(* Logix 5000 project; controller Tekno_ASRS vendor 1 type 14 code 147 rev 20.11; software revision 20.01; part 3 of 4 *)
(* tags used below, declared in another part *)
   AutoMode : BOOL;
   AAxis : AXIS_CIP_DRIVE;
   AAxisJog : MOTION_INSTRUCTION;
   AAxisMAM : MOTION_INSTRUCTION;
   AAxisMove : BOOL;
   AAxisOn : MOTION_INSTRUCTION;
   AAxisSODelay : TIMER;
   AAxisStop : MOTION_INSTRUCTION;
   ABayPos : DINT;
   ABGrid : Position[100,20];
   AgridLoc : DINT;
   AGVatDP : ALIAS FOR StationaryIO:1:I.3;
   AGVatPU : ALIAS FOR StationaryIO:1:I.2;
   AGVDP : BOOL;
   AGVok2LvDP : ALIAS FOR StationaryIO:8:O.0;
   AGVok2LvPU : ALIAS FOR StationaryIO:8:O.1;
   AGVPU : BOOL;
   AGVPUHoldTmr : TIMER;
   AInc : DINT;
   AllowSynchAB : BOOL;
   APitch : REAL;
   APos : REAL;
   ARange : REAL;
   AReq : DINT;
   AReqPos : REAL;
   ASRSMCR : BOOL;
   AStart : REAL;
   BAxis : AXIS_CIP_DRIVE;
   BAxisJog : MOTION_INSTRUCTION;
   BAxisMAM : MOTION_INSTRUCTION;
   BAxisMove : BOOL;
   BAxisOn : MOTION_INSTRUCTION;
   BAxisSODelay : TIMER;
   BAxisStop : MOTION_INSTRUCTION;
   BBayPos : DINT;
   BgridLoc : DINT;
   BInc : DINT;
   BPitch : REAL;
   BPos : REAL;
   BRange : DINT;
   BReq : DINT;
   BReqPos : REAL;
   BStart : REAL;
   CCoordSetup : BOOL;
   CfgEnd : BayPos;
   CfgStrt : BayPos;
   CfgTtlAAxis : DINT;
   CfgTtlBAxis : DINT;
   CFinalPos : DINT;
   CGridLoc : DINT;
   CHomePos : DINT;
   Configuration : Configuration;
   CPosHighLim : DINT;
   CPosLowLim : DINT;
   CPosSpeed2Tol : DINT;
   CPosTolerance : DINT;
   CReq : DINT;
   CReqPos : DINT;
   CurrentAPos : DINT;
   CurrentBPos : DINT;
   CurrentCPos : DINT;
   CurrentTask : Task;
   DepositReq : BOOL;
   FootSwitch : ALIAS FOR ShuttleIO:9:I.Pt04Data;
   HMI_Commands : HMI_Commands;
   HomeSpatula : BOOL;
   JogAAxisEn : BOOL;
   JogActive : BOOL;
   JogARev : BOOL;
   JogBAxisEn : BOOL;
   JogBFwd : BOOL;
   JogBRev : BOOL;
   JogConfiguration : Configuration;
   JogEnabled : BOOL;
   JogReleaseSBrk : BOOL;
   Last : DINT;
   LastAAxErr : DINT;
   LastAAxExErr : DINT;
   LastMessageReceiveSequence : DINT;
   LoadTask : Task;
   LockRelease : ALIAS FOR StationaryIO:7:I.Pt04Data;
   ManOnBoard : ALIAS FOR ShuttleIO:5:O.5;
   MatrixSetup : BOOL;
   MaxA : DINT;
   MaxB : DINT;
   MoveComplete : BOOL;
   MoveInProcess : BOOL;
   MoveReady : BOOL;
   MoveRequested : BOOL;
   MoveSafetyEnable : BOOL;
   MsgTimer : TIMER;
   MtrEndDsbleZn : REAL;
   OperatorDN : BOOL;
   PnlEndDsbleZn : REAL;
   PorDInProc : BOOL;
   PorDStepTemp : BOOL;
   PorDStop : BOOL;
   PositionFlt : BOOL;
   ReceiveMessage : Messaging;
   ReleaseSpatBrk : BOOL;
   SendMessage : Messaging;
   SendMessageCommand : MESSAGE;
   SpatSimHome : BOOL;
   SpatulaBrake : ALIAS FOR ShuttleIO:5:O.6;
   SpatulaExtendComp : BOOL;
   SpatulaExtended : BOOL;
   SpatulaHome : ALIAS FOR ShuttleIO:2:I.4;
   SpatulaStopped : BOOL;
   SUIndPos : BOOL;
   TaskFIFO : CONTROL;
   TaskFile : Task[100];
   TaskInProcess : BOOL;
   TestStop : BOOL;
   XAccuracy : REAL;
   XAxisMtrSideEOT : ALIAS FOR ShuttleIO:2:I.6;
   XAxisPnlSideEOT : ALIAS FOR ShuttleIO:2:I.7;
   XHighLimit : REAL;
   XLftTempDint1 : DINT;
   XLftTempDint2 : DINT;
   XLftTempFloat1 : REAL;
   XLftTempFloat2 : REAL;
   XLftTempFloat3 : REAL;
   XLowLimit : REAL;
   XRgtTempDint1 : DINT;
   XRgtTempDint2 : REAL;
   XRgtTempFloat1 : REAL;
   XRgtTempFloat2 : REAL;
   XRgtTempFloat3 : REAL;
   XStCalMode : ALIAS FOR StationaryIO:5:O.Data[0].0;
   XStLftSignRun : ALIAS FOR StationaryIO:5:I.Data[7].7;
   XStrain : Strain;
   XStrainHigh : DINT;
   XStrainLow : DINT;
   XStRtSignRun : ALIAS FOR StationaryIO:5:I.Data[11].7;
   XStRunMode : ALIAS FOR StationaryIO:5:O.Data[0].1;
   XTensionOK : BOOL;
   ZAccuracy : REAL;
   ZAxisDnEOT : ALIAS FOR ShuttleIO:1:I.1;
   ZAxisUpEOT : ALIAS FOR ShuttleIO:1:I.0;
   ZForeStCalMode : ALIAS FOR ShuttleIO:3:O.Data[0].0;
   ZForeStrain : Strain;
   ZForeStRunMode : ALIAS FOR ShuttleIO:3:O.Data[0].1;
   ZHighLimit : REAL;
   ZLBindTmr : TIMER;
   ZLFault : BOOL;
   ZLowLimit : REAL;
   ZLsDisengaged : BOOL;
(* MainProgram, continued *)

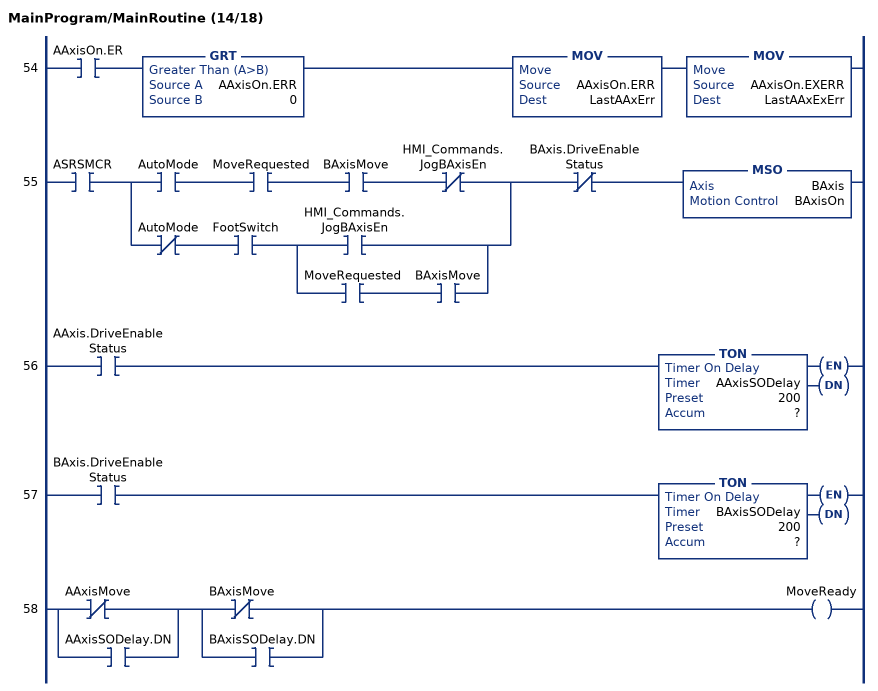
   [picture p24: MainProgram/MainRoutine rungs 54-58]
   54: XIC(AAxisOn.ER)GRT(AAxisOn.ERR,0)MOV(AAxisOn.ERR,LastAAxErr)MOV(AAxisOn.EXERR,LastAAxExErr);
   55: XIC(ASRSMCR)[XIC(AutoMode) XIC(MoveRequested) XIC(BAxisMove) XIO(HMI_Commands.JogBAxisEn) ,XIO(AutoMode) XIC(FootSwitch) [XIC(HMI_Commands.JogBAxisEn) ,XIC(MoveRequested) XIC(BAxisMove) ] ]XIO(BAxis.DriveEnableStatus)MSO(BAxis,BAxisOn);
   56: XIC(AAxis.DriveEnableStatus)TON(AAxisSODelay,?,?);
   57: XIC(BAxis.DriveEnableStatus)TON(BAxisSODelay,?,?);
   58: [XIO(AAxisMove) ,XIC(AAxisSODelay.DN) ][XIO(BAxisMove) ,XIC(BAxisSODelay.DN) ]OTE(MoveReady);
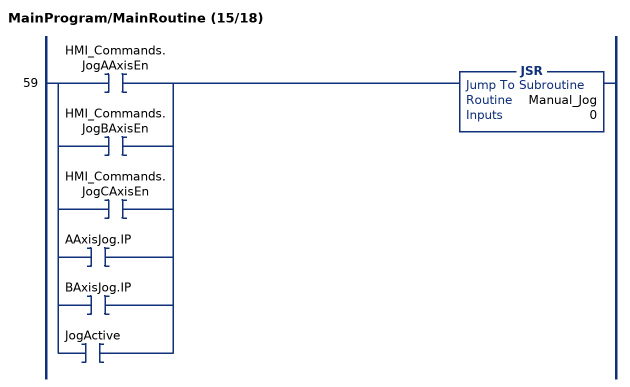
   59: [XIC(HMI_Commands.JogAAxisEn) ,XIC(HMI_Commands.JogBAxisEn) ,XIC(HMI_Commands.JogCAxisEn) ,XIC(AAxisJog.IP) ,XIC(BAxisJog.IP) ,XIC(JogActive) ]JSR(Manual_Jog,0);
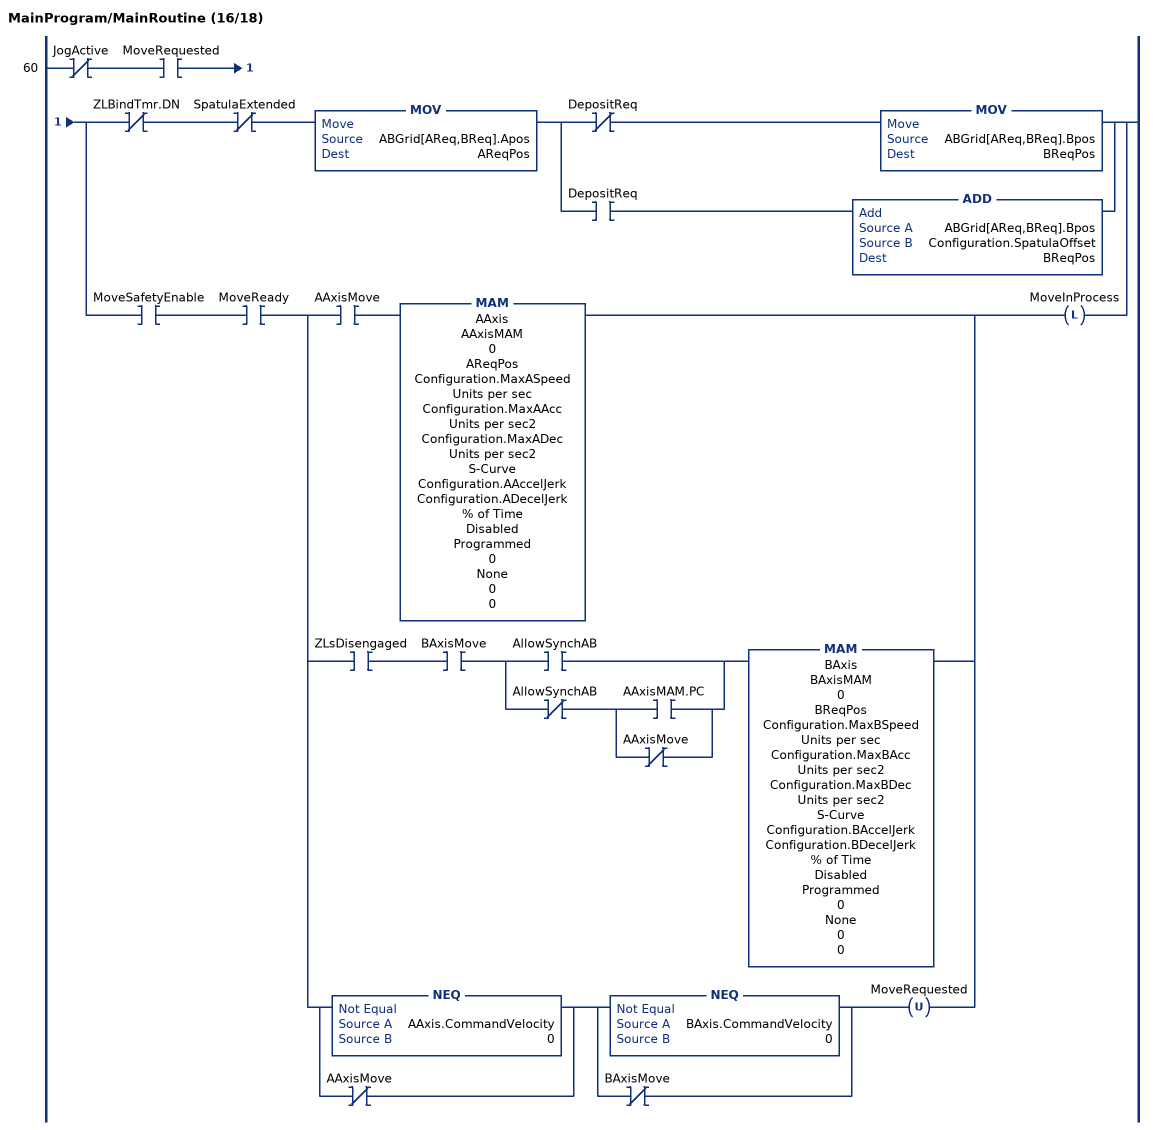
   60: XIO(JogActive)XIC(MoveRequested)[XIO(ZLBindTmr.DN) XIO(SpatulaExtended) MOV(ABGrid[AReq,BReq].Apos,AReqPos) [XIO(DepositReq) MOV(ABGrid[AReq,BReq].Bpos,BReqPos) ,XIC(DepositReq) ADD(ABGrid[AReq,BReq].Bpos,Configuration.SpatulaOffset,BReqPos) ] ,XIC(MoveSafetyEnable) XIC(MoveReady) [XIC(AAxisMove) MAM(AAxis,AAxisMAM,0,AReqPos,Configuration.MaxASpeed,Units per sec,Configuration.MaxAAcc,Units per sec2,Configuration.MaxADec,Units per sec2,S-Curve,Configuration.AAccelJerk,Configuration.ADecelJerk,% of Time,Disabled,Programmed,0,None,0,0) ,XIC(ZLsDisengaged) XIC(BAxisMove) [XIC(AllowSynchAB) ,XIO(AllowSynchAB) [XIC(AAxisMAM.PC) ,XIO(AAxisMove) ] ] MAM(BAxis,BAxisMAM,0,BReqPos,Configuration.MaxBSpeed,Units per sec,Configuration.MaxBAcc,Units per sec2,Configuration.MaxBDec,Units per sec2,S-Curve,Configuration.BAccelJerk,Configuration.BDecelJerk,% of Time,Disabled,Programmed,0,None,0,0) ,[NEQ(AAxis.CommandVelocity,0) ,XIO(AAxisMove) ] [NEQ(BAxis.CommandVelocity,0) ,XIO(BAxisMove) ] OTU(MoveRequested) ] OTL(MoveInProcess) ];
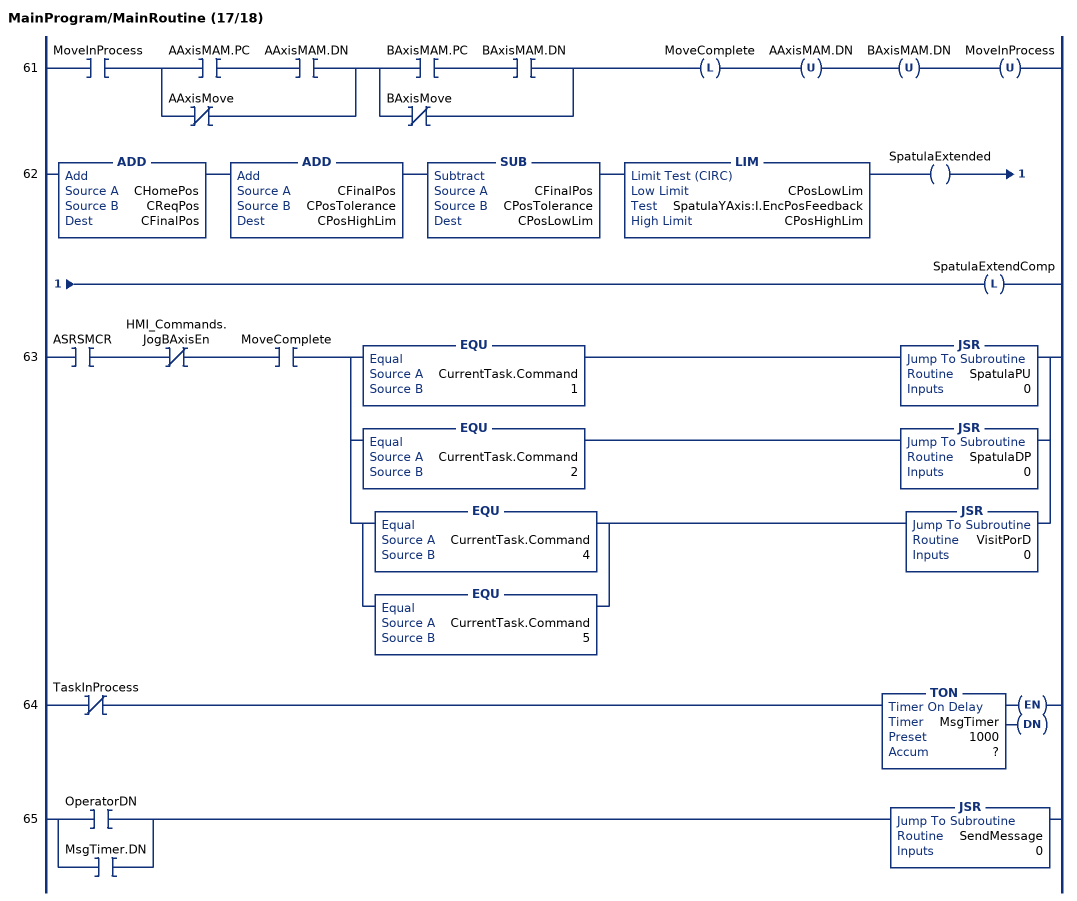
   61: XIC(MoveInProcess)[XIC(AAxisMAM.PC) XIC(AAxisMAM.DN) ,XIO(AAxisMove) ][XIC(BAxisMAM.PC) XIC(BAxisMAM.DN) ,XIO(BAxisMove) ]OTL(MoveComplete)OTU(AAxisMAM.DN)OTU(BAxisMAM.DN)OTU(MoveInProcess);
   62: ADD(CHomePos,CReqPos,CFinalPos)ADD(CFinalPos,CPosTolerance,CPosHighLim)SUB(CFinalPos,CPosTolerance,CPosLowLim)LIM(CPosLowLim,SpatulaYAxis:I.EncPosFeedback,CPosHighLim)OTE(SpatulaExtended)OTL(SpatulaExtendComp);
   63: XIC(ASRSMCR)XIO(HMI_Commands.JogBAxisEn)XIC(MoveComplete)[EQU(CurrentTask.Command,1) JSR(SpatulaPU,0) ,EQU(CurrentTask.Command,2) JSR(SpatulaDP,0) ,[EQU(CurrentTask.Command,4) ,EQU(CurrentTask.Command,5) ] JSR(VisitPorD,0) ];
   64: XIO(TaskInProcess)TON(MsgTimer,?,?);
   65: [XIC(OperatorDN) ,XIC(MsgTimer.DN) ]JSR(SendMessage,0);
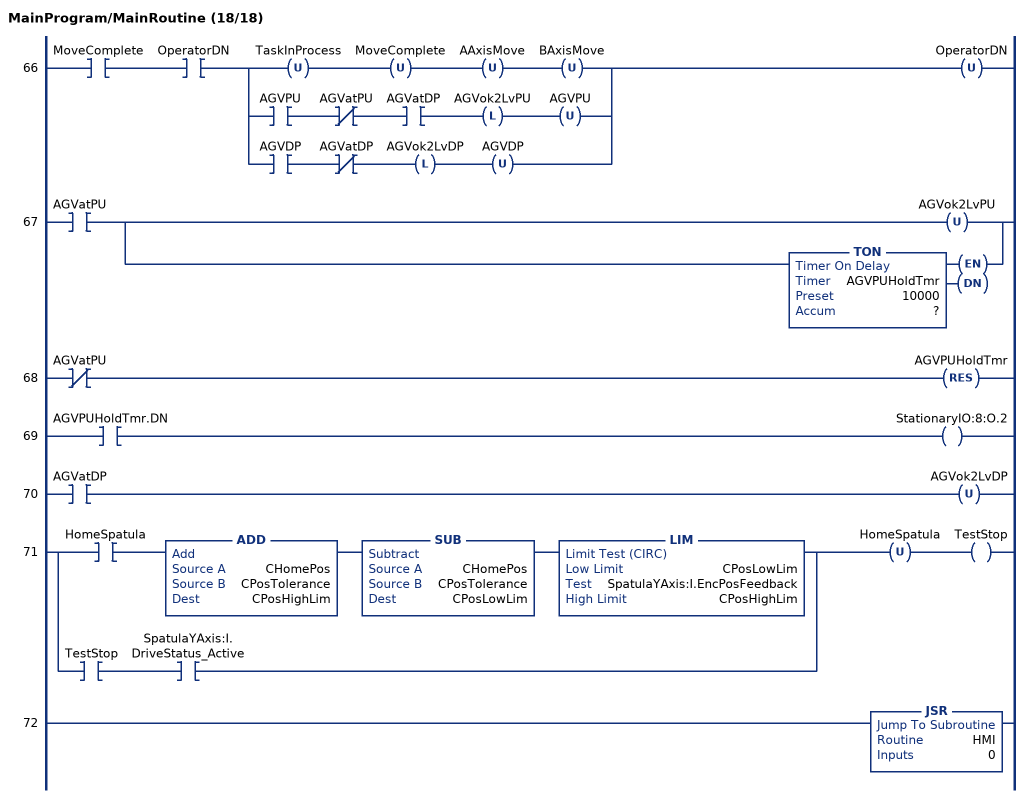
   66: XIC(MoveComplete)XIC(OperatorDN)[OTU(TaskInProcess) OTU(MoveComplete) OTU(AAxisMove) OTU(BAxisMove) ,XIC(AGVPU) XIO(AGVatPU) XIC(AGVatDP) OTL(AGVok2LvPU) OTU(AGVPU) ,XIC(AGVDP) XIO(AGVatDP) OTL(AGVok2LvDP) OTU(AGVDP) ]OTU(OperatorDN);
   67: XIC(AGVatPU)[OTU(AGVok2LvPU) ,TON(AGVPUHoldTmr,?,?) ];
   68: XIO(AGVatPU)RES(AGVPUHoldTmr);
   69: XIC(AGVPUHoldTmr.DN)OTE(StationaryIO:8:O.2);
   70: XIC(AGVatDP)OTU(AGVok2LvDP);
   71: [XIC(HomeSpatula) ADD(CHomePos,CPosTolerance,CPosHighLim) SUB(CHomePos,CPosTolerance,CPosLowLim) LIM(CPosLowLim,SpatulaYAxis:I.EncPosFeedback,CPosHighLim) ,XIC(TestStop) XIC(SpatulaYAxis:I.DriveStatus_Active) ]OTU(HomeSpatula)OTE(TestStop);
   72: JSR(HMI,0);
END_ROUTINE

ROUTINE Manual_Jog   (* ladder *)
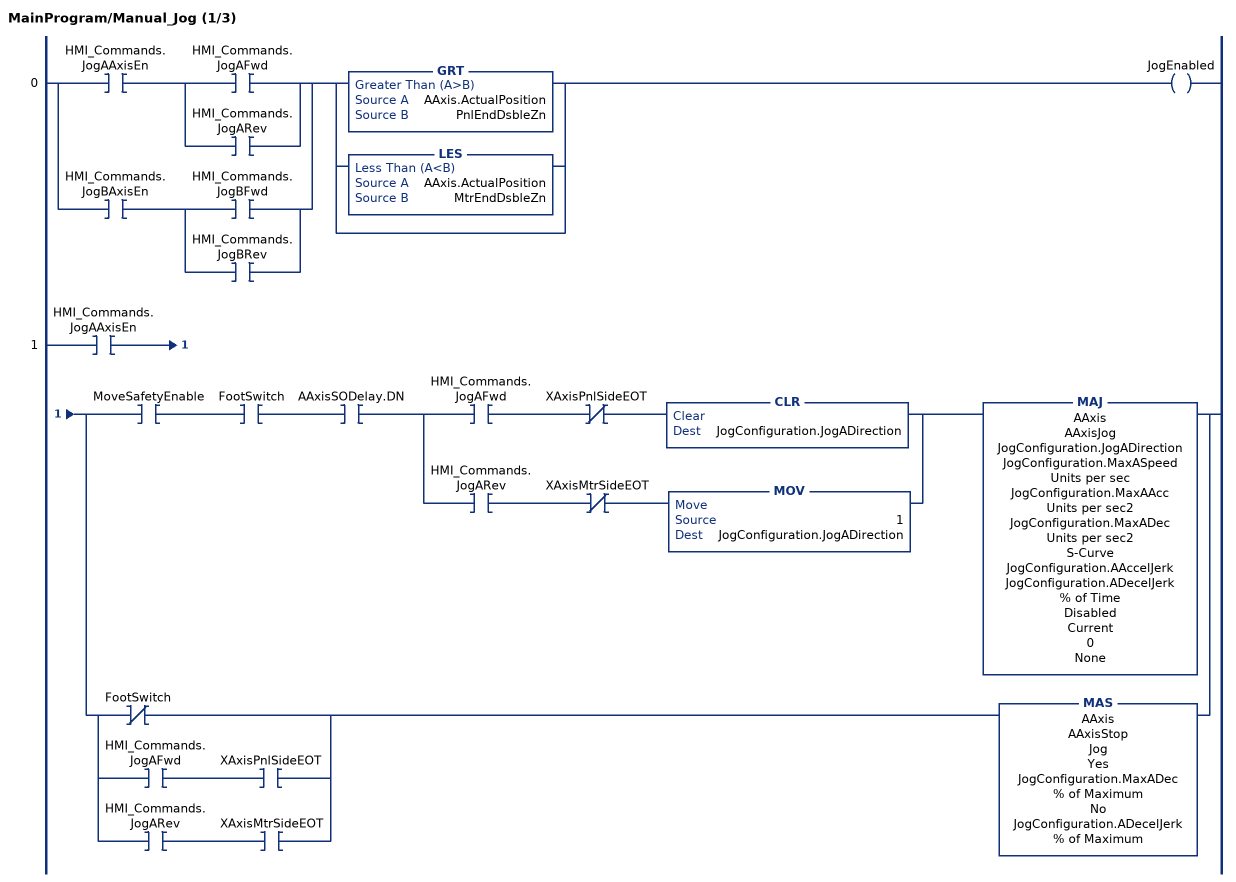
   0: [XIC(HMI_Commands.JogAAxisEn) [XIC(HMI_Commands.JogAFwd) ,XIC(HMI_Commands.JogARev) ] ,XIC(HMI_Commands.JogBAxisEn) [XIC(HMI_Commands.JogBFwd) ,XIC(HMI_Commands.JogBRev) ] ][GRT(AAxis.ActualPosition,PnlEndDsbleZn) ,LES(AAxis.ActualPosition,MtrEndDsbleZn) ,]OTE(JogEnabled);
   1: XIC(HMI_Commands.JogAAxisEn)[XIC(MoveSafetyEnable) XIC(FootSwitch) XIC(AAxisSODelay.DN) [XIC(HMI_Commands.JogAFwd) XIO(XAxisPnlSideEOT) CLR(JogConfiguration.JogADirection) ,XIC(HMI_Commands.JogARev) XIO(XAxisMtrSideEOT) MOV(1,JogConfiguration.JogADirection) ] MAJ(AAxis,AAxisJog,JogConfiguration.JogADirection,JogConfiguration.MaxASpeed,Units per sec,JogConfiguration.MaxAAcc,Units per sec2,JogConfiguration.MaxADec,Units per sec2,S-Curve,JogConfiguration.AAccelJerk,JogConfiguration.ADecelJerk,% of Time,Disabled,Current,0,None) ,[XIO(FootSwitch) ,XIC(HMI_Commands.JogAFwd) XIC(XAxisPnlSideEOT) ,XIC(HMI_Commands.JogARev) XIC(XAxisMtrSideEOT) ] MAS(AAxis,AAxisStop,Jog,Yes,JogConfiguration.MaxADec,% of Maximum,No,JogConfiguration.ADecelJerk,% of Maximum) ];
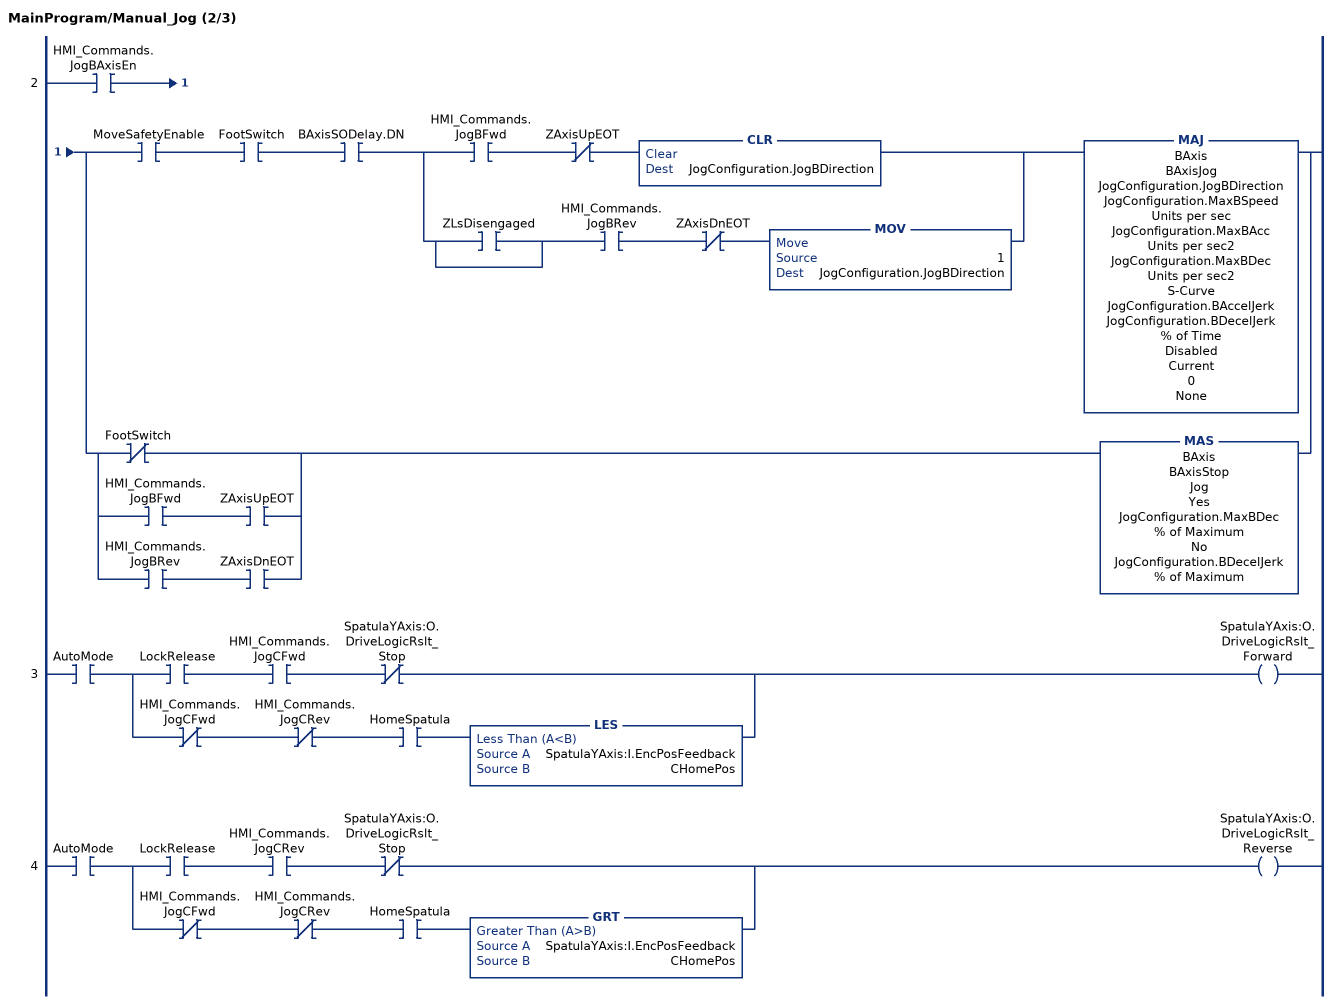
   2: XIC(HMI_Commands.JogBAxisEn)[XIC(MoveSafetyEnable) XIC(FootSwitch) XIC(BAxisSODelay.DN) [XIC(HMI_Commands.JogBFwd) XIO(ZAxisUpEOT) CLR(JogConfiguration.JogBDirection) ,[XIC(ZLsDisengaged) ,] XIC(HMI_Commands.JogBRev) XIO(ZAxisDnEOT) MOV(1,JogConfiguration.JogBDirection) ] MAJ(BAxis,BAxisJog,JogConfiguration.JogBDirection,JogConfiguration.MaxBSpeed,Units per sec,JogConfiguration.MaxBAcc,Units per sec2,JogConfiguration.MaxBDec,Units per sec2,S-Curve,JogConfiguration.BAccelJerk,JogConfiguration.BDecelJerk,% of Time,Disabled,Current,0,None) ,[XIO(FootSwitch) ,XIC(HMI_Commands.JogBFwd) XIC(ZAxisUpEOT) ,XIC(HMI_Commands.JogBRev) XIC(ZAxisDnEOT) ] MAS(BAxis,BAxisStop,Jog,Yes,JogConfiguration.MaxBDec,% of Maximum,No,JogConfiguration.BDecelJerk,% of Maximum) ];
   3: XIC(AutoMode)[XIC(LockRelease) XIC(HMI_Commands.JogCFwd) XIO(SpatulaYAxis:O.DriveLogicRslt_Stop) ,XIO(HMI_Commands.JogCFwd) XIO(HMI_Commands.JogCRev) XIC(HomeSpatula) LES(SpatulaYAxis:I.EncPosFeedback,CHomePos) ]OTE(SpatulaYAxis:O.DriveLogicRslt_Forward);
   4: XIC(AutoMode)[XIC(LockRelease) XIC(HMI_Commands.JogCRev) XIO(SpatulaYAxis:O.DriveLogicRslt_Stop) ,XIO(HMI_Commands.JogCFwd) XIO(HMI_Commands.JogCRev) XIC(HomeSpatula) GRT(SpatulaYAxis:I.EncPosFeedback,CHomePos) ]OTE(SpatulaYAxis:O.DriveLogicRslt_Reverse);
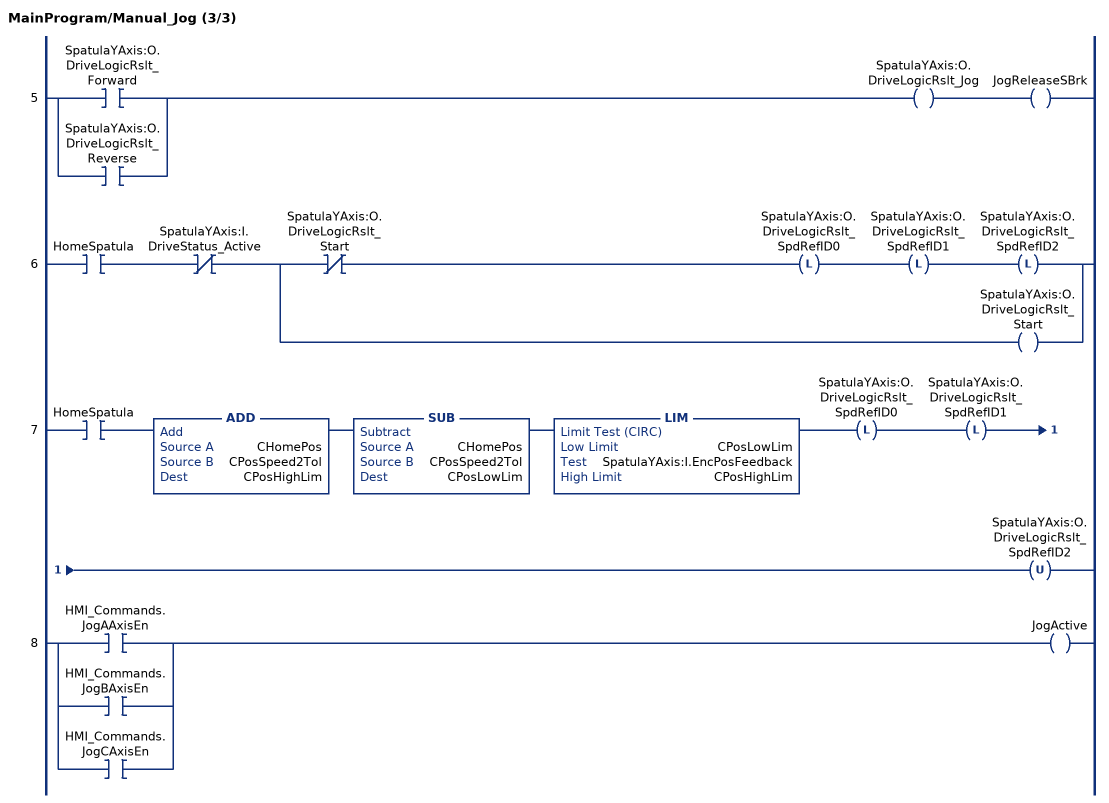
   5: [XIC(SpatulaYAxis:O.DriveLogicRslt_Forward) ,XIC(SpatulaYAxis:O.DriveLogicRslt_Reverse) ]OTE(SpatulaYAxis:O.DriveLogicRslt_Jog)OTE(JogReleaseSBrk);
   6: XIC(HomeSpatula)XIO(SpatulaYAxis:I.DriveStatus_Active)[XIO(SpatulaYAxis:O.DriveLogicRslt_Start) OTL(SpatulaYAxis:O.DriveLogicRslt_SpdRefID0) OTL(SpatulaYAxis:O.DriveLogicRslt_SpdRefID1) OTL(SpatulaYAxis:O.DriveLogicRslt_SpdRefID2) ,OTE(SpatulaYAxis:O.DriveLogicRslt_Start) ];
   7: XIC(HomeSpatula)ADD(CHomePos,CPosSpeed2Tol,CPosHighLim)SUB(CHomePos,CPosSpeed2Tol,CPosLowLim)LIM(CPosLowLim,SpatulaYAxis:I.EncPosFeedback,CPosHighLim)OTL(SpatulaYAxis:O.DriveLogicRslt_SpdRefID0)OTL(SpatulaYAxis:O.DriveLogicRslt_SpdRefID1)OTU(SpatulaYAxis:O.DriveLogicRslt_SpdRefID2);
   8: [XIC(HMI_Commands.JogAAxisEn) ,XIC(HMI_Commands.JogBAxisEn) ,XIC(HMI_Commands.JogCAxisEn) ]OTE(JogActive);
END_ROUTINE

ROUTINE ReceiveMessage   (* ladder *)
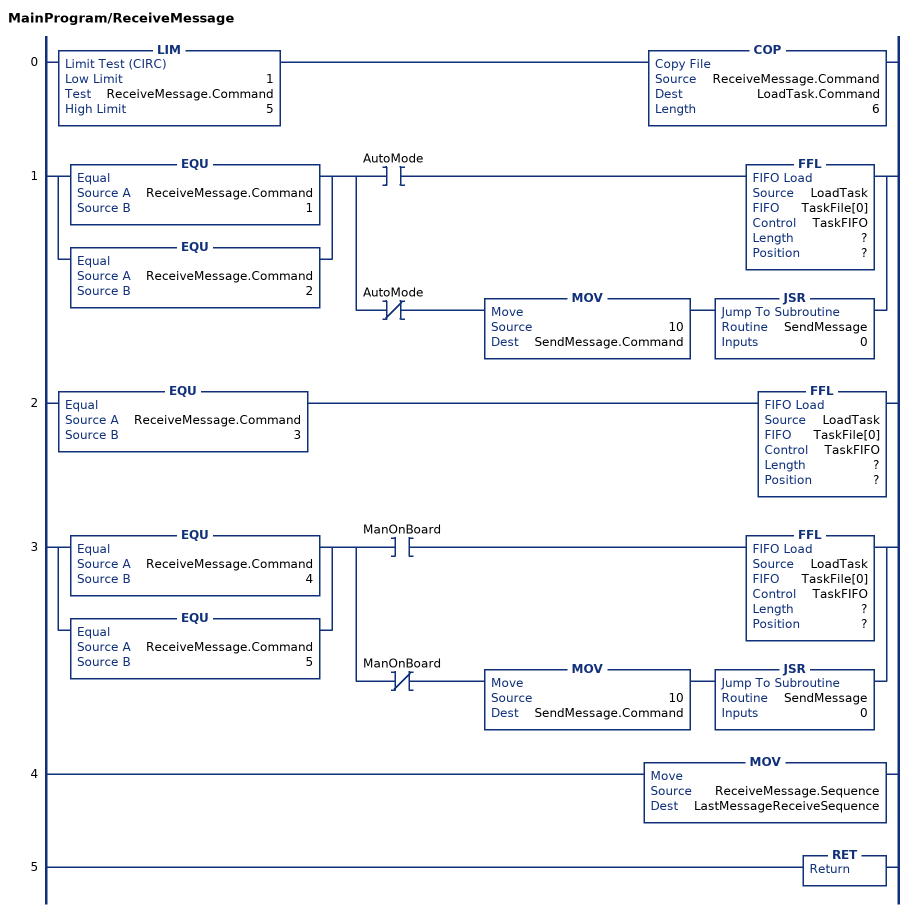
   0: LIM(1,ReceiveMessage.Command,5)COP(ReceiveMessage.Command,LoadTask.Command,6);
   1: [EQU(ReceiveMessage.Command,1) ,EQU(ReceiveMessage.Command,2) ][XIC(AutoMode) FFL(LoadTask,TaskFile[0],TaskFIFO,?,?) ,XIO(AutoMode) MOV(10,SendMessage.Command) JSR(SendMessage,0) ];
   2: EQU(ReceiveMessage.Command,3)FFL(LoadTask,TaskFile[0],TaskFIFO,?,?);
   3: [EQU(ReceiveMessage.Command,4) ,EQU(ReceiveMessage.Command,5) ][XIC(ManOnBoard) FFL(LoadTask,TaskFile[0],TaskFIFO,?,?) ,XIO(ManOnBoard) MOV(10,SendMessage.Command) JSR(SendMessage,0) ];
   4: MOV(ReceiveMessage.Sequence,LastMessageReceiveSequence);
   5: RET();
END_ROUTINE

ROUTINE SendMessage   (* ladder *)
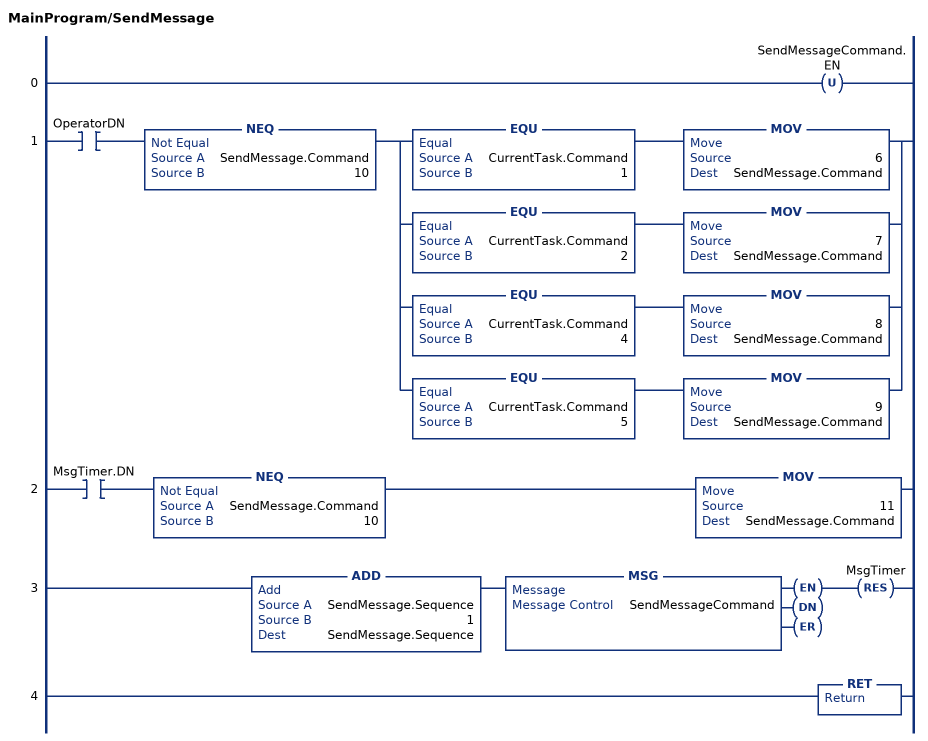
   0: OTU(SendMessageCommand.EN);
   1: XIC(OperatorDN)NEQ(SendMessage.Command,10)[EQU(CurrentTask.Command,1) MOV(6,SendMessage.Command) ,EQU(CurrentTask.Command,2) MOV(7,SendMessage.Command) ,EQU(CurrentTask.Command,4) MOV(8,SendMessage.Command) ,EQU(CurrentTask.Command,5) MOV(9,SendMessage.Command) ];
   2: XIC(MsgTimer.DN)NEQ(SendMessage.Command,10)MOV(11,SendMessage.Command);
   3: ADD(SendMessage.Sequence,1,SendMessage.Sequence)MSG(SendMessageCommand)RES(MsgTimer);
   4: RET();
END_ROUTINE

ROUTINE Setup   (* ladder *)
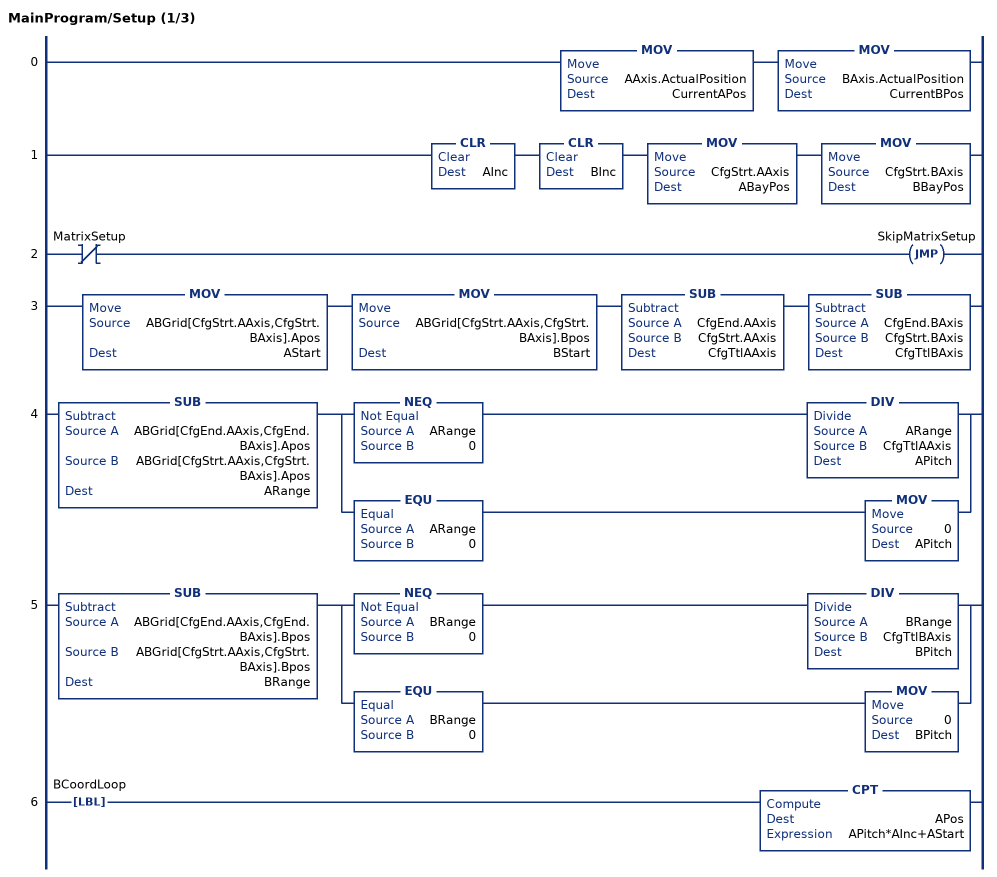
   0: MOV(AAxis.ActualPosition,CurrentAPos)MOV(BAxis.ActualPosition,CurrentBPos);
   1: CLR(AInc)CLR(BInc)MOV(CfgStrt.AAxis,ABayPos)MOV(CfgStrt.BAxis,BBayPos);
   2: XIO(MatrixSetup)JMP(SkipMatrixSetup);
   3: MOV(ABGrid[CfgStrt.AAxis,CfgStrt.BAxis].Apos,AStart)MOV(ABGrid[CfgStrt.AAxis,CfgStrt.BAxis].Bpos,BStart)SUB(CfgEnd.AAxis,CfgStrt.AAxis,CfgTtlAAxis)SUB(CfgEnd.BAxis,CfgStrt.BAxis,CfgTtlBAxis);
   4: SUB(ABGrid[CfgEnd.AAxis,CfgEnd.BAxis].Apos,ABGrid[CfgStrt.AAxis,CfgStrt.BAxis].Apos,ARange)[NEQ(ARange,0) DIV(ARange,CfgTtlAAxis,APitch) ,EQU(ARange,0) MOV(0,APitch) ];
   5: SUB(ABGrid[CfgEnd.AAxis,CfgEnd.BAxis].Bpos,ABGrid[CfgStrt.AAxis,CfgStrt.BAxis].Bpos,BRange)[NEQ(BRange,0) DIV(BRange,CfgTtlBAxis,BPitch) ,EQU(BRange,0) MOV(0,BPitch) ];
   6: LBL(BCoordLoop)CPT(APos,APitch*AInc+AStart);
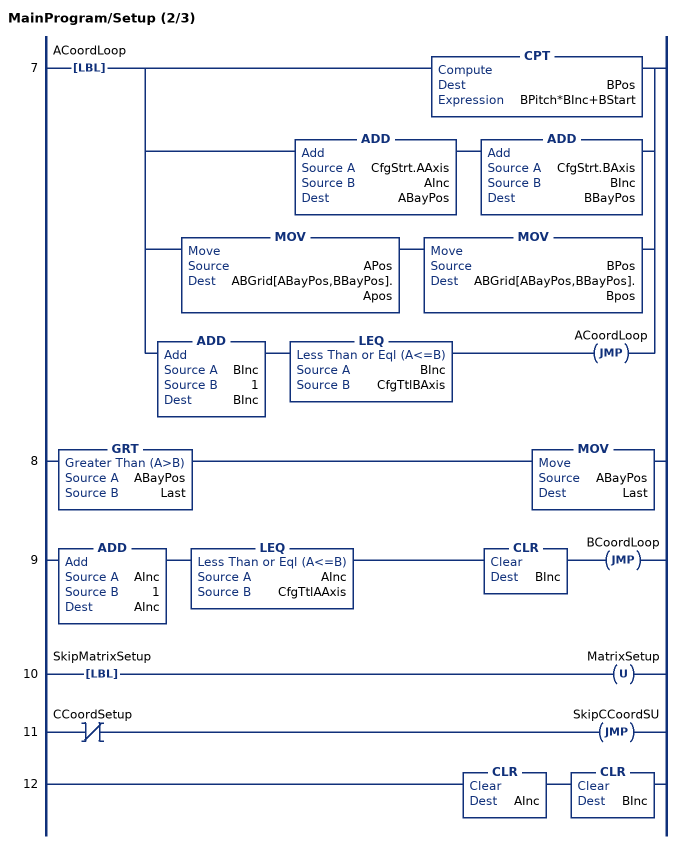
   7: LBL(ACoordLoop)[CPT(BPos,BPitch*BInc+BStart) ,ADD(CfgStrt.AAxis,AInc,ABayPos) ADD(CfgStrt.BAxis,BInc,BBayPos) ,MOV(APos,ABGrid[ABayPos,BBayPos].Apos) MOV(BPos,ABGrid[ABayPos,BBayPos].Bpos) ,ADD(BInc,1,BInc) LEQ(BInc,CfgTtlBAxis) JMP(ACoordLoop) ];
   8: GRT(ABayPos,Last)MOV(ABayPos,Last);
   9: ADD(AInc,1,AInc)LEQ(AInc,CfgTtlAAxis)CLR(BInc)JMP(BCoordLoop);
   10: LBL(SkipMatrixSetup)OTU(MatrixSetup);
   11: XIO(CCoordSetup)JMP(SkipCCoordSU);
   12: CLR(AInc)CLR(BInc);
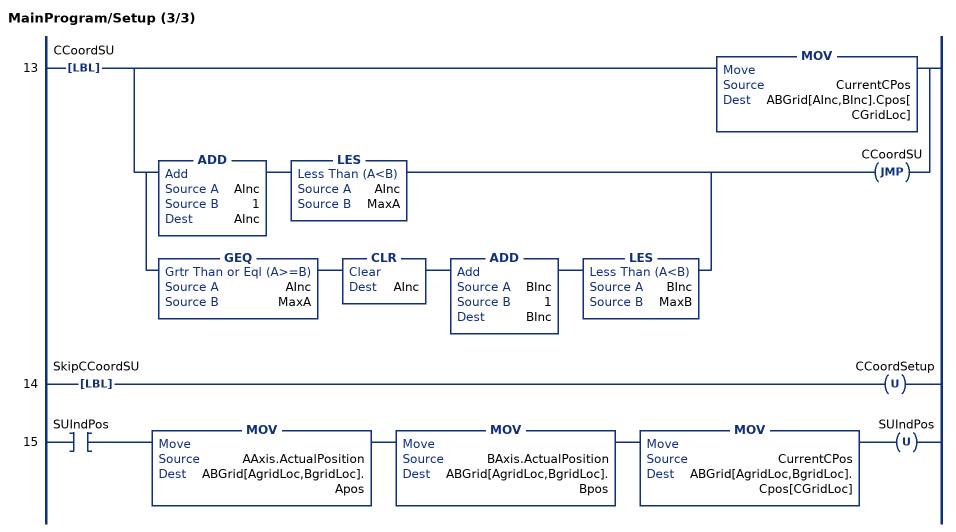
   13: LBL(CCoordSU)[MOV(CurrentCPos,ABGrid[AInc,BInc].Cpos[CGridLoc]) ,[ADD(AInc,1,AInc) LES(AInc,MaxA) ,GEQ(AInc,MaxA) CLR(AInc) ADD(BInc,1,BInc) LES(BInc,MaxB) ] JMP(CCoordSU) ];
   14: LBL(SkipCCoordSU)OTU(CCoordSetup);
   15: XIC(SUIndPos)MOV(AAxis.ActualPosition,ABGrid[AgridLoc,BgridLoc].Apos)MOV(BAxis.ActualPosition,ABGrid[AgridLoc,BgridLoc].Bpos)MOV(CurrentCPos,ABGrid[AgridLoc,BgridLoc].Cpos[CGridLoc])OTU(SUIndPos);
END_ROUTINE

ROUTINE SpatulaDP   (* ladder *)
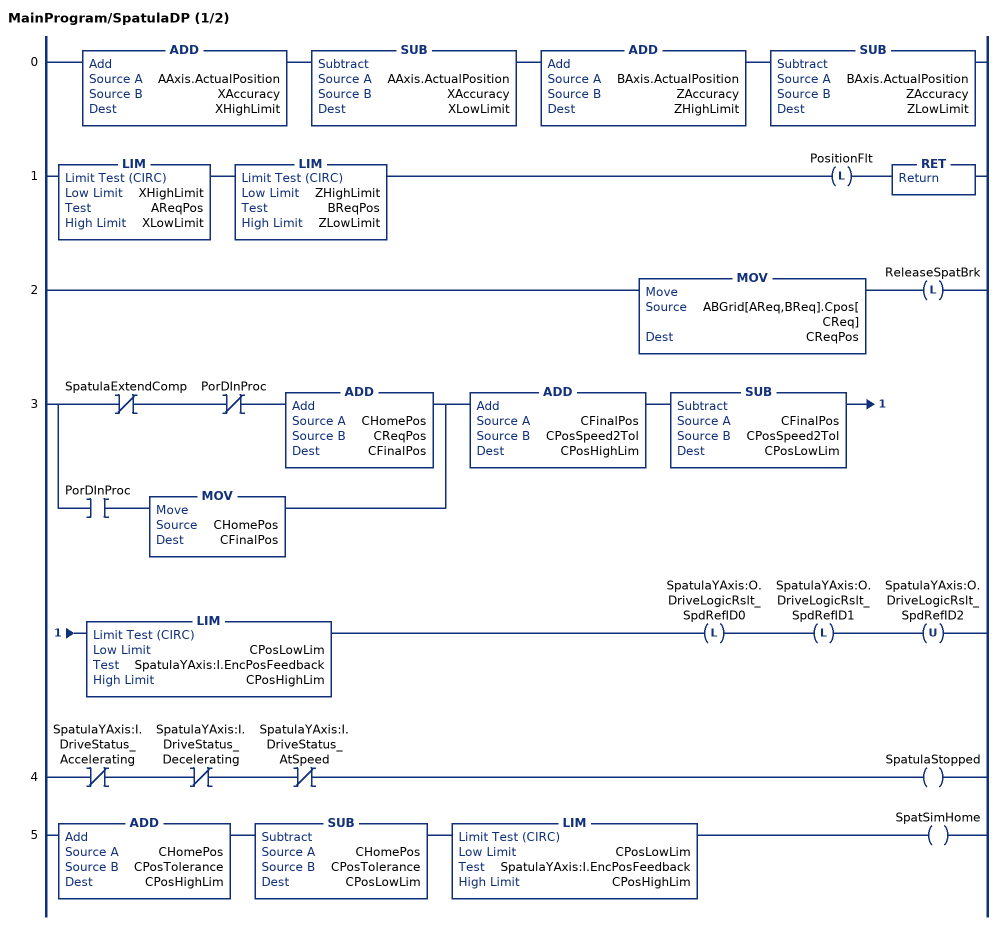
   0: ADD(AAxis.ActualPosition,XAccuracy,XHighLimit)SUB(AAxis.ActualPosition,XAccuracy,XLowLimit)ADD(BAxis.ActualPosition,ZAccuracy,ZHighLimit)SUB(BAxis.ActualPosition,ZAccuracy,ZLowLimit);
   1: LIM(XHighLimit,AReqPos,XLowLimit)LIM(ZHighLimit,BReqPos,ZLowLimit)OTL(PositionFlt)RET();
   2: MOV(ABGrid[AReq,BReq].Cpos[CReq],CReqPos)OTL(ReleaseSpatBrk);
   3: [XIO(SpatulaExtendComp) XIO(PorDInProc) ADD(CHomePos,CReqPos,CFinalPos) ,XIC(PorDInProc) MOV(CHomePos,CFinalPos) ]ADD(CFinalPos,CPosSpeed2Tol,CPosHighLim)SUB(CFinalPos,CPosSpeed2Tol,CPosLowLim)LIM(CPosLowLim,SpatulaYAxis:I.EncPosFeedback,CPosHighLim)OTL(SpatulaYAxis:O.DriveLogicRslt_SpdRefID0)OTL(SpatulaYAxis:O.DriveLogicRslt_SpdRefID1)OTU(SpatulaYAxis:O.DriveLogicRslt_SpdRefID2);
   4: XIO(SpatulaYAxis:I.DriveStatus_Accelerating)XIO(SpatulaYAxis:I.DriveStatus_Decelerating)XIO(SpatulaYAxis:I.DriveStatus_AtSpeed)OTE(SpatulaStopped);
   5: ADD(CHomePos,CPosTolerance,CPosHighLim)SUB(CHomePos,CPosTolerance,CPosLowLim)LIM(CPosLowLim,SpatulaYAxis:I.EncPosFeedback,CPosHighLim)OTE(SpatSimHome);
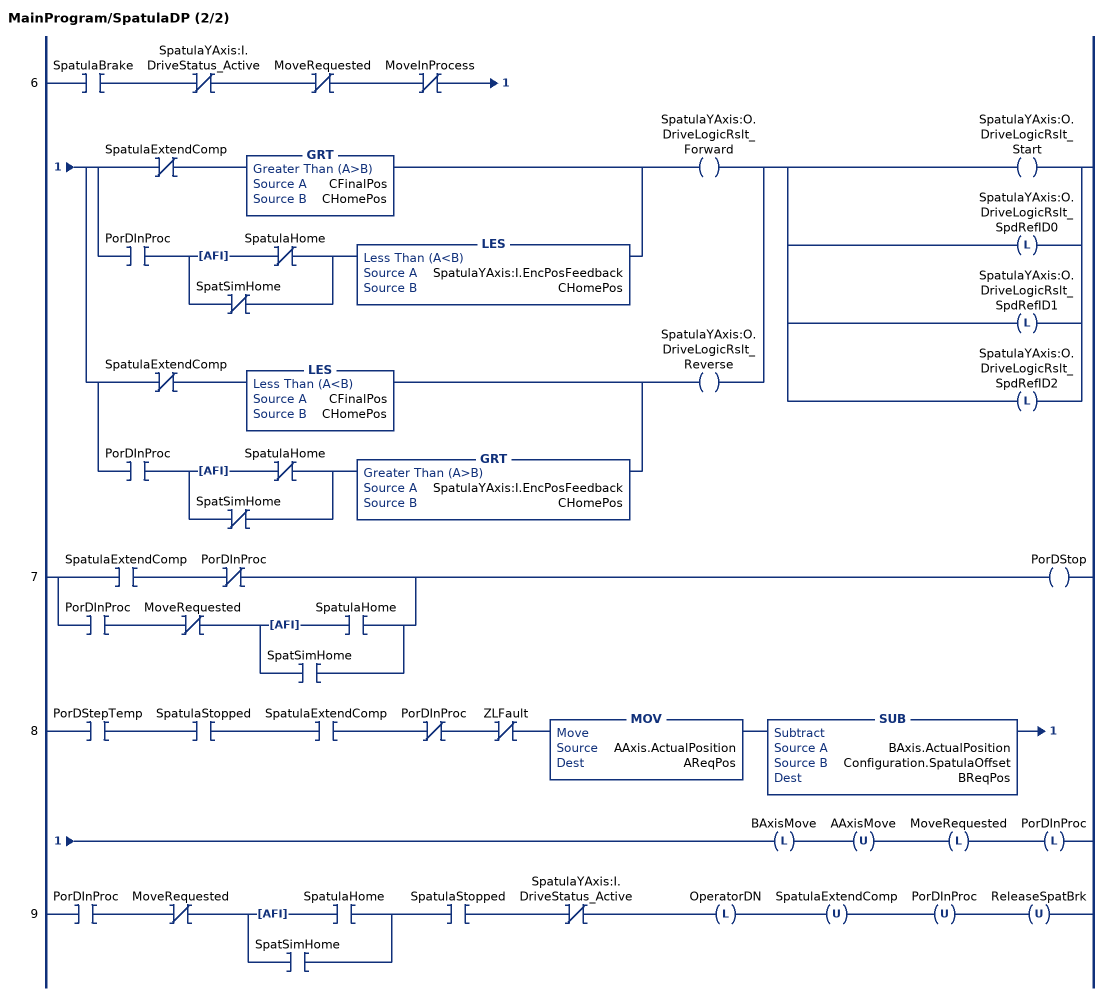
   6: XIC(SpatulaBrake)XIO(SpatulaYAxis:I.DriveStatus_Active)XIO(MoveRequested)XIO(MoveInProcess)[[XIO(SpatulaExtendComp) GRT(CFinalPos,CHomePos) ,XIC(PorDInProc) [AFI() XIO(SpatulaHome) ,XIO(SpatSimHome) ] LES(SpatulaYAxis:I.EncPosFeedback,CHomePos) ] OTE(SpatulaYAxis:O.DriveLogicRslt_Forward) ,[XIO(SpatulaExtendComp) LES(CFinalPos,CHomePos) ,XIC(PorDInProc) [AFI() XIO(SpatulaHome) ,XIO(SpatSimHome) ] GRT(SpatulaYAxis:I.EncPosFeedback,CHomePos) ] OTE(SpatulaYAxis:O.DriveLogicRslt_Reverse) ][OTE(SpatulaYAxis:O.DriveLogicRslt_Start) ,OTL(SpatulaYAxis:O.DriveLogicRslt_SpdRefID0) ,OTL(SpatulaYAxis:O.DriveLogicRslt_SpdRefID1) ,OTL(SpatulaYAxis:O.DriveLogicRslt_SpdRefID2) ];
   7: [XIC(SpatulaExtendComp) XIO(PorDInProc) ,XIC(PorDInProc) XIO(MoveRequested) [AFI() XIC(SpatulaHome) ,XIC(SpatSimHome) ] ]OTE(PorDStop);
   8: XIC(PorDStepTemp)XIC(SpatulaStopped)XIC(SpatulaExtendComp)XIO(PorDInProc)XIO(ZLFault)MOV(AAxis.ActualPosition,AReqPos)SUB(BAxis.ActualPosition,Configuration.SpatulaOffset,BReqPos)OTL(BAxisMove)OTU(AAxisMove)OTL(MoveRequested)OTL(PorDInProc);
   9: XIC(PorDInProc)XIO(MoveRequested)[AFI() XIC(SpatulaHome) ,XIC(SpatSimHome) ]XIC(SpatulaStopped)XIO(SpatulaYAxis:I.DriveStatus_Active)OTL(OperatorDN)OTU(SpatulaExtendComp)OTU(PorDInProc)OTU(ReleaseSpatBrk);
END_ROUTINE

ROUTINE SpatulaPU   (* ladder *)
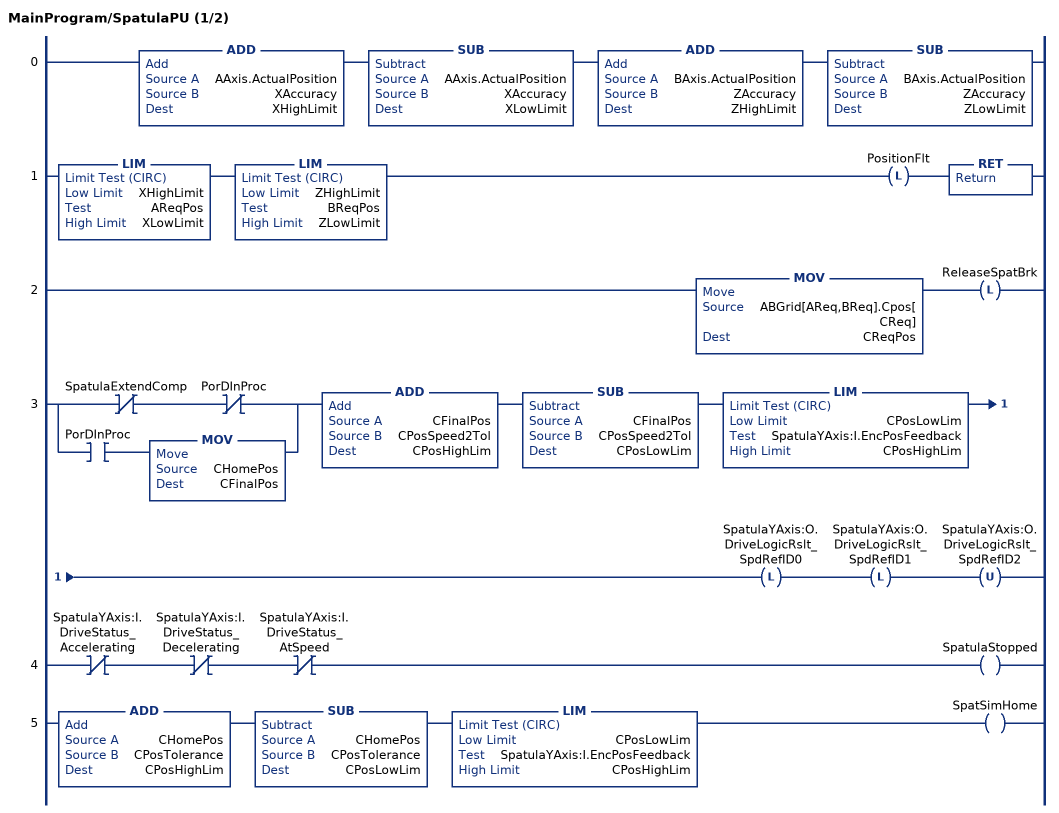
   0: ADD(AAxis.ActualPosition,XAccuracy,XHighLimit)SUB(AAxis.ActualPosition,XAccuracy,XLowLimit)ADD(BAxis.ActualPosition,ZAccuracy,ZHighLimit)SUB(BAxis.ActualPosition,ZAccuracy,ZLowLimit);
   1: LIM(XHighLimit,AReqPos,XLowLimit)LIM(ZHighLimit,BReqPos,ZLowLimit)OTL(PositionFlt)RET();
   2: MOV(ABGrid[AReq,BReq].Cpos[CReq],CReqPos)OTL(ReleaseSpatBrk);
   3: [XIO(SpatulaExtendComp) XIO(PorDInProc) ,XIC(PorDInProc) MOV(CHomePos,CFinalPos) ]ADD(CFinalPos,CPosSpeed2Tol,CPosHighLim)SUB(CFinalPos,CPosSpeed2Tol,CPosLowLim)LIM(CPosLowLim,SpatulaYAxis:I.EncPosFeedback,CPosHighLim)OTL(SpatulaYAxis:O.DriveLogicRslt_SpdRefID0)OTL(SpatulaYAxis:O.DriveLogicRslt_SpdRefID1)OTU(SpatulaYAxis:O.DriveLogicRslt_SpdRefID2);
   4: XIO(SpatulaYAxis:I.DriveStatus_Accelerating)XIO(SpatulaYAxis:I.DriveStatus_Decelerating)XIO(SpatulaYAxis:I.DriveStatus_AtSpeed)OTE(SpatulaStopped);
   5: ADD(CHomePos,CPosTolerance,CPosHighLim)SUB(CHomePos,CPosTolerance,CPosLowLim)LIM(CPosLowLim,SpatulaYAxis:I.EncPosFeedback,CPosHighLim)OTE(SpatSimHome);
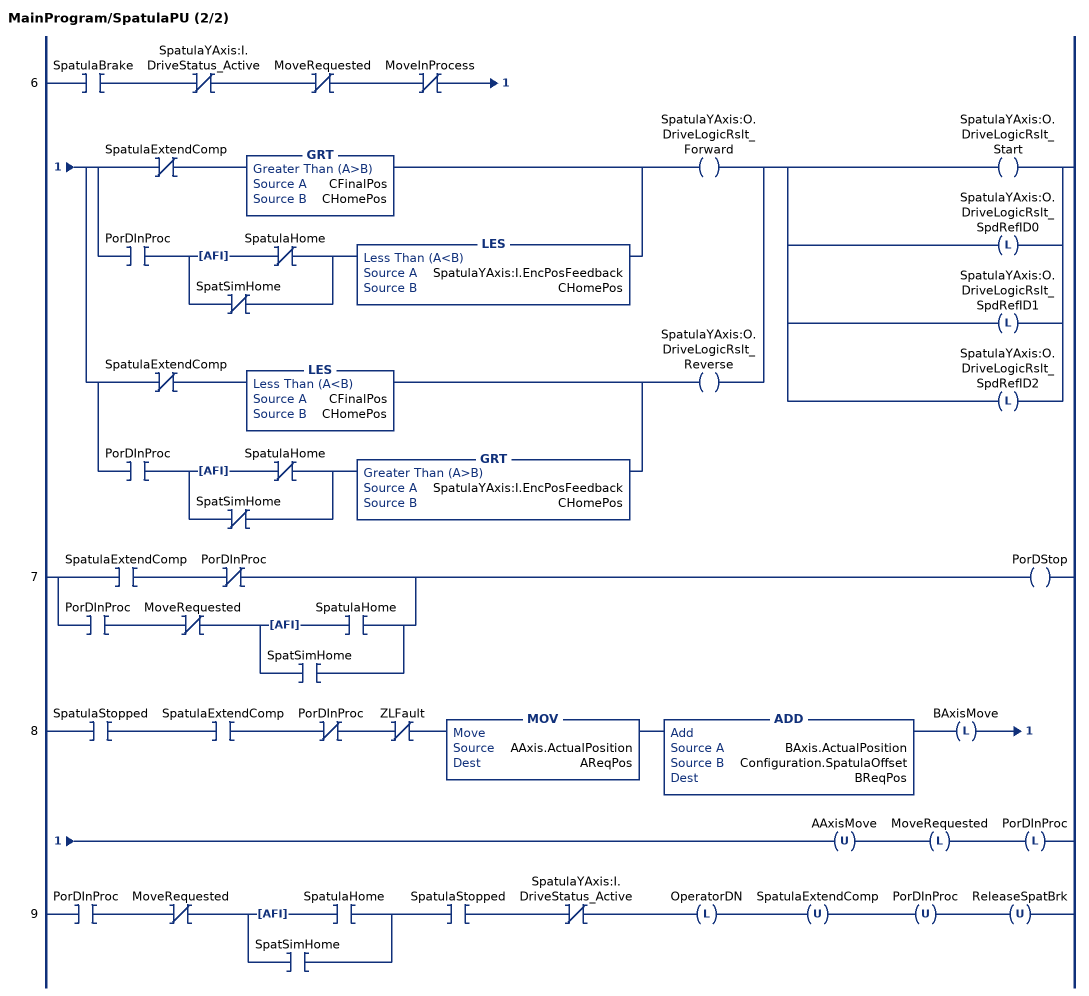
   6: XIC(SpatulaBrake)XIO(SpatulaYAxis:I.DriveStatus_Active)XIO(MoveRequested)XIO(MoveInProcess)[[XIO(SpatulaExtendComp) GRT(CFinalPos,CHomePos) ,XIC(PorDInProc) [AFI() XIO(SpatulaHome) ,XIO(SpatSimHome) ] LES(SpatulaYAxis:I.EncPosFeedback,CHomePos) ] OTE(SpatulaYAxis:O.DriveLogicRslt_Forward) ,[XIO(SpatulaExtendComp) LES(CFinalPos,CHomePos) ,XIC(PorDInProc) [AFI() XIO(SpatulaHome) ,XIO(SpatSimHome) ] GRT(SpatulaYAxis:I.EncPosFeedback,CHomePos) ] OTE(SpatulaYAxis:O.DriveLogicRslt_Reverse) ][OTE(SpatulaYAxis:O.DriveLogicRslt_Start) ,OTL(SpatulaYAxis:O.DriveLogicRslt_SpdRefID0) ,OTL(SpatulaYAxis:O.DriveLogicRslt_SpdRefID1) ,OTL(SpatulaYAxis:O.DriveLogicRslt_SpdRefID2) ];
   7: [XIC(SpatulaExtendComp) XIO(PorDInProc) ,XIC(PorDInProc) XIO(MoveRequested) [AFI() XIC(SpatulaHome) ,XIC(SpatSimHome) ] ]OTE(PorDStop);
   8: XIC(SpatulaStopped)XIC(SpatulaExtendComp)XIO(PorDInProc)XIO(ZLFault)MOV(AAxis.ActualPosition,AReqPos)ADD(BAxis.ActualPosition,Configuration.SpatulaOffset,BReqPos)OTL(BAxisMove)OTU(AAxisMove)OTL(MoveRequested)OTL(PorDInProc);
   9: XIC(PorDInProc)XIO(MoveRequested)[AFI() XIC(SpatulaHome) ,XIC(SpatSimHome) ]XIC(SpatulaStopped)XIO(SpatulaYAxis:I.DriveStatus_Active)OTL(OperatorDN)OTU(SpatulaExtendComp)OTU(PorDInProc)OTU(ReleaseSpatBrk);
END_ROUTINE

ROUTINE StrainGauges   (* ladder *)
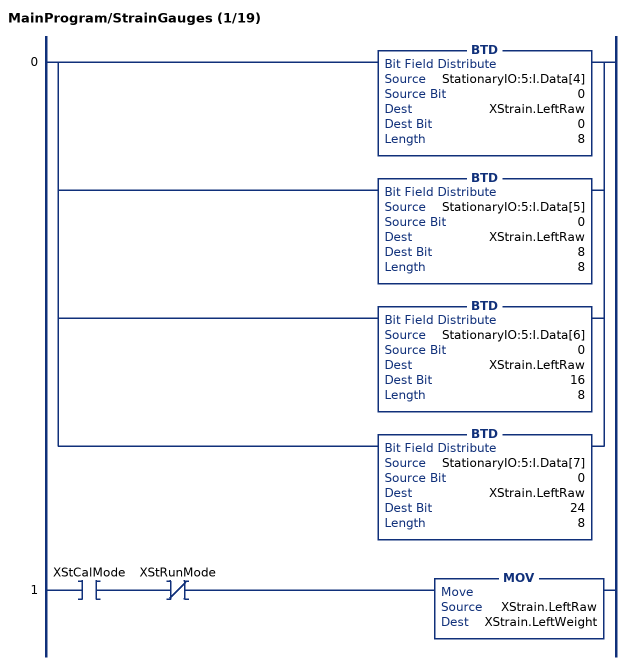
   0: [BTD(StationaryIO:5:I.Data[4],0,XStrain.LeftRaw,0,8) ,BTD(StationaryIO:5:I.Data[5],0,XStrain.LeftRaw,8,8) ,BTD(StationaryIO:5:I.Data[6],0,XStrain.LeftRaw,16,8) ,BTD(StationaryIO:5:I.Data[7],0,XStrain.LeftRaw,24,8) ];
   1: XIC(XStCalMode)XIO(XStRunMode)MOV(XStrain.LeftRaw,XStrain.LeftWeight);
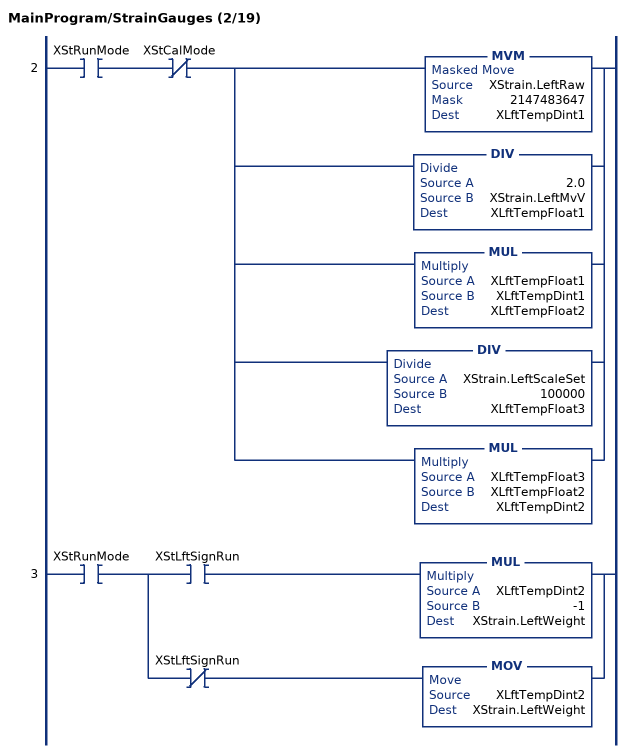
   2: XIC(XStRunMode)XIO(XStCalMode)[MVM(XStrain.LeftRaw,2147483647,XLftTempDint1) ,DIV(2.0,XStrain.LeftMvV,XLftTempFloat1) ,MUL(XLftTempFloat1,XLftTempDint1,XLftTempFloat2) ,DIV(XStrain.LeftScaleSet,100000,XLftTempFloat3) ,MUL(XLftTempFloat3,XLftTempFloat2,XLftTempDint2) ];
   3: XIC(XStRunMode)[XIC(XStLftSignRun) MUL(XLftTempDint2,-1,XStrain.LeftWeight) ,XIO(XStLftSignRun) MOV(XLftTempDint2,XStrain.LeftWeight) ];
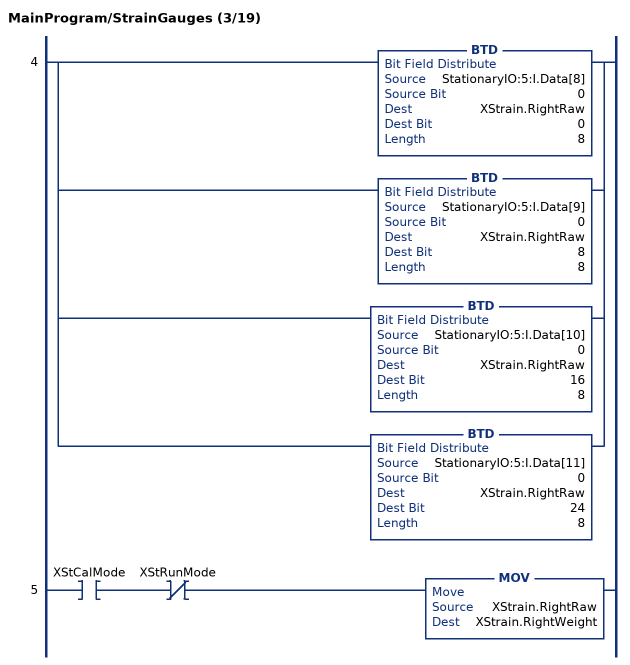
   4: [BTD(StationaryIO:5:I.Data[8],0,XStrain.RightRaw,0,8) ,BTD(StationaryIO:5:I.Data[9],0,XStrain.RightRaw,8,8) ,BTD(StationaryIO:5:I.Data[10],0,XStrain.RightRaw,16,8) ,BTD(StationaryIO:5:I.Data[11],0,XStrain.RightRaw,24,8) ];
   5: XIC(XStCalMode)XIO(XStRunMode)MOV(XStrain.RightRaw,XStrain.RightWeight);
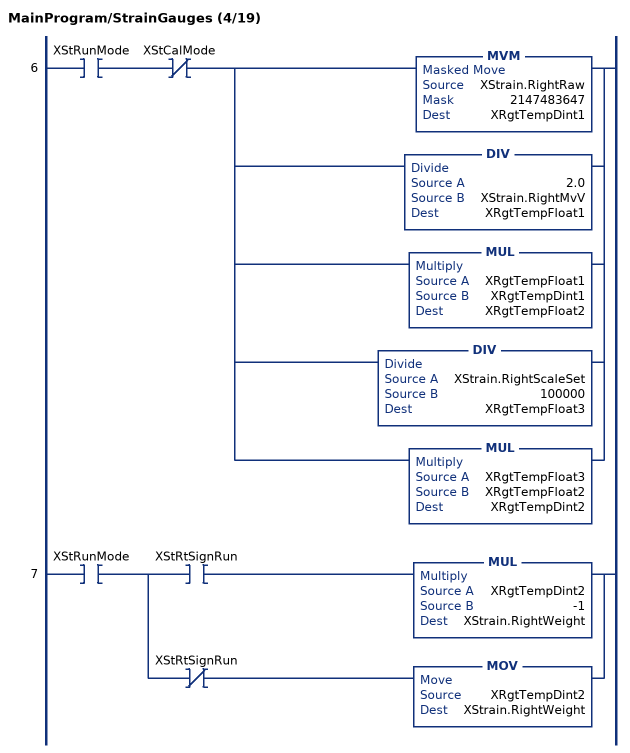
   6: XIC(XStRunMode)XIO(XStCalMode)[MVM(XStrain.RightRaw,2147483647,XRgtTempDint1) ,DIV(2.0,XStrain.RightMvV,XRgtTempFloat1) ,MUL(XRgtTempFloat1,XRgtTempDint1,XRgtTempFloat2) ,DIV(XStrain.RightScaleSet,100000,XRgtTempFloat3) ,MUL(XRgtTempFloat3,XRgtTempFloat2,XRgtTempDint2) ];
   7: XIC(XStRunMode)[XIC(XStRtSignRun) MUL(XRgtTempDint2,-1,XStrain.RightWeight) ,XIO(XStRtSignRun) MOV(XRgtTempDint2,XStrain.RightWeight) ];
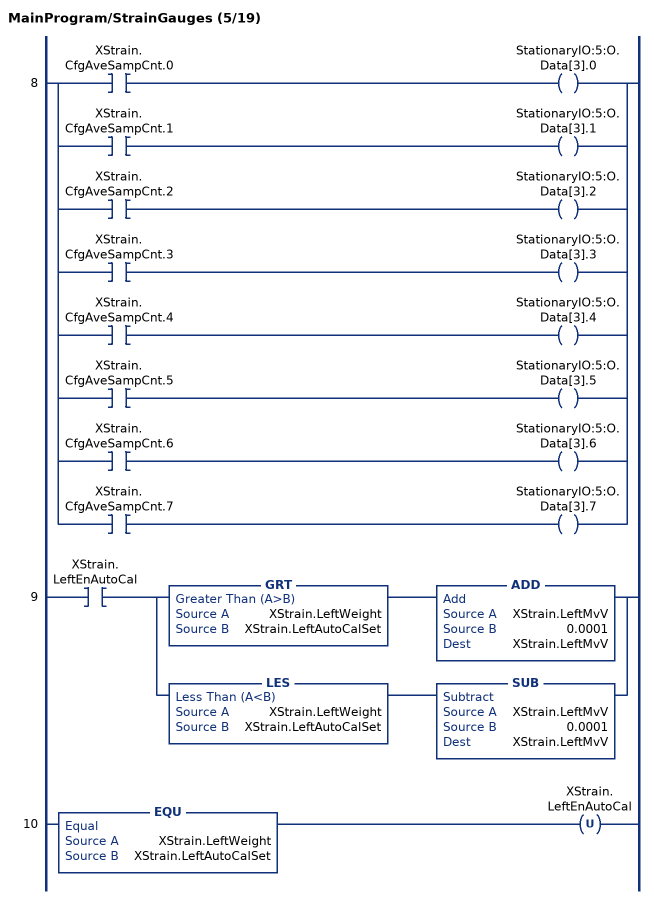
   8: [XIC(XStrain.CfgAveSampCnt.0) OTE(StationaryIO:5:O.Data[3].0) ,XIC(XStrain.CfgAveSampCnt.1) OTE(StationaryIO:5:O.Data[3].1) ,XIC(XStrain.CfgAveSampCnt.2) OTE(StationaryIO:5:O.Data[3].2) ,XIC(XStrain.CfgAveSampCnt.3) OTE(StationaryIO:5:O.Data[3].3) ,XIC(XStrain.CfgAveSampCnt.4) OTE(StationaryIO:5:O.Data[3].4) ,XIC(XStrain.CfgAveSampCnt.5) OTE(StationaryIO:5:O.Data[3].5) ,XIC(XStrain.CfgAveSampCnt.6) OTE(StationaryIO:5:O.Data[3].6) ,XIC(XStrain.CfgAveSampCnt.7) OTE(StationaryIO:5:O.Data[3].7) ];
   9: XIC(XStrain.LeftEnAutoCal)[GRT(XStrain.LeftWeight,XStrain.LeftAutoCalSet) ADD(XStrain.LeftMvV,0.0001,XStrain.LeftMvV) ,LES(XStrain.LeftWeight,XStrain.LeftAutoCalSet) SUB(XStrain.LeftMvV,0.0001,XStrain.LeftMvV) ];
   10: EQU(XStrain.LeftWeight,XStrain.LeftAutoCalSet)OTU(XStrain.LeftEnAutoCal);
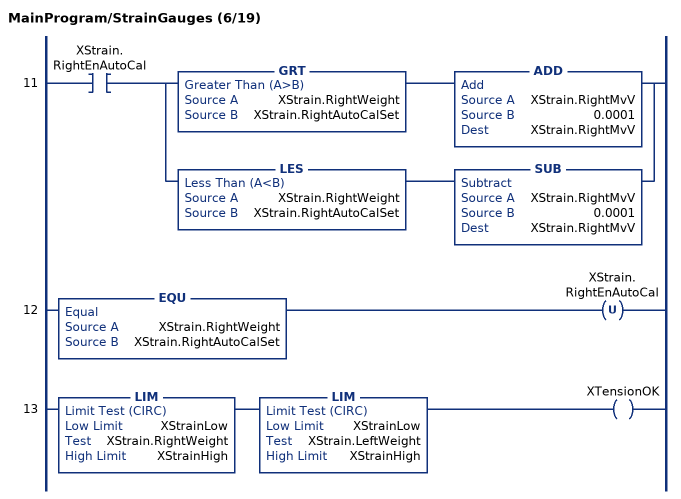
   11: XIC(XStrain.RightEnAutoCal)[GRT(XStrain.RightWeight,XStrain.RightAutoCalSet) ADD(XStrain.RightMvV,0.0001,XStrain.RightMvV) ,LES(XStrain.RightWeight,XStrain.RightAutoCalSet) SUB(XStrain.RightMvV,0.0001,XStrain.RightMvV) ];
   12: EQU(XStrain.RightWeight,XStrain.RightAutoCalSet)OTU(XStrain.RightEnAutoCal);
   13: LIM(XStrainLow,XStrain.RightWeight,XStrainHigh)LIM(XStrainLow,XStrain.LeftWeight,XStrainHigh)OTE(XTensionOK);
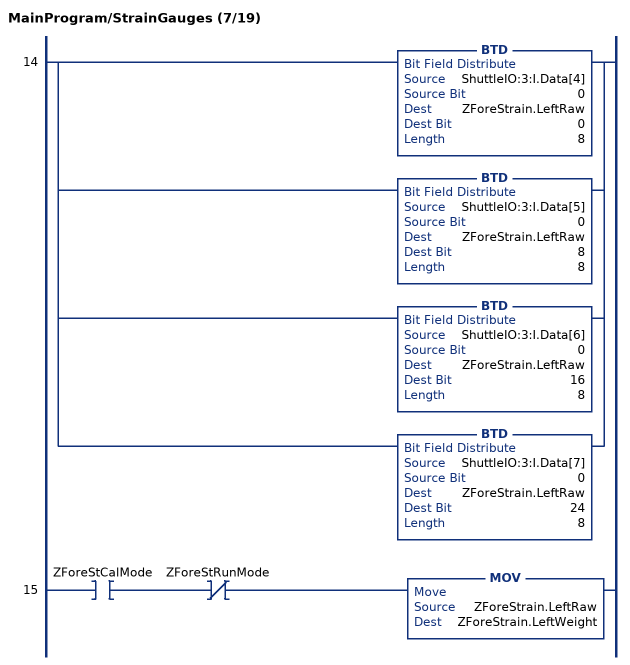
   14: [BTD(ShuttleIO:3:I.Data[4],0,ZForeStrain.LeftRaw,0,8) ,BTD(ShuttleIO:3:I.Data[5],0,ZForeStrain.LeftRaw,8,8) ,BTD(ShuttleIO:3:I.Data[6],0,ZForeStrain.LeftRaw,16,8) ,BTD(ShuttleIO:3:I.Data[7],0,ZForeStrain.LeftRaw,24,8) ];
   15: XIC(ZForeStCalMode)XIO(ZForeStRunMode)MOV(ZForeStrain.LeftRaw,ZForeStrain.LeftWeight);
